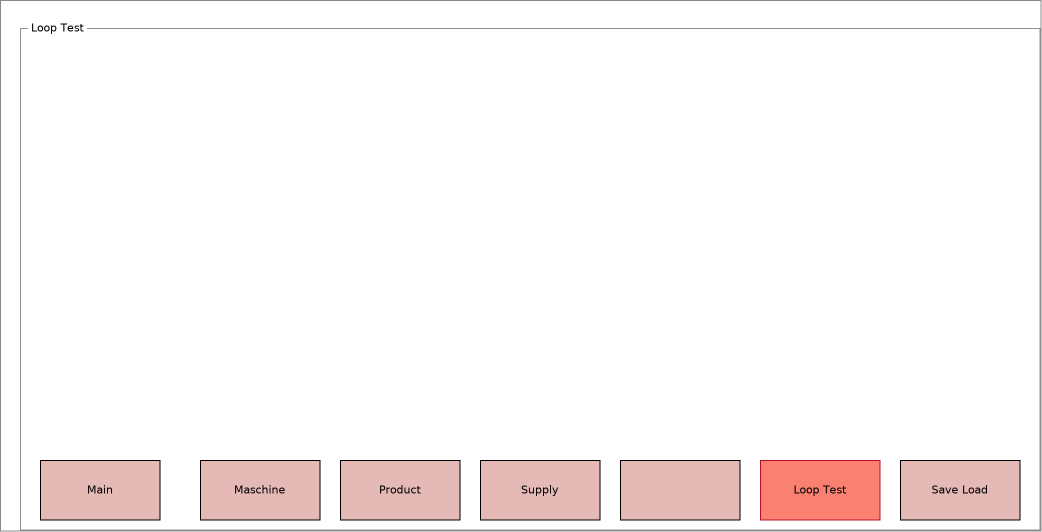
VISUALIZATION Visu_LoopTest  // 1042x532
    GroupBox (20,20 1020x510), "Loop Test"
        Rectangle (20,440 120x60), "Main"
            OnMouseClick: change screen: Visu_Main
        Rectangle (880,440 120x60), "Save Load"
            OnMouseClick: change screen: Visu_SaveLoad
        Rectangle (320,440 120x60), "Product"
            OnMouseClick: change screen: Visu_PParam
        Rectangle (180,440 120x60), "Maschine"
            OnMouseClick: change screen: Visu_MParam
        Rectangle (460,440 120x60), "Supply"
            OnMouseClick: change screen: Visu_Supply
        Rectangle (600,440 120x60)
        Rectangle (740,440 120x60), "Loop Test"
            OnMouseClick: change screen: Visu_LoopTest
END_VISUALIZATION

(* stored: Version 1.1.0.1, ProductVersion 3.1.4024.12
   Visu Visu_LoopTest: Id {72b28d07-ecb1-4681-abf7-47095e70440c} *)
